# EPICS substitutions: ek9000App/Db/EL2004.substitutions
file EL2004.template
{       pattern
        {
                TERMINAL,

        }
        {
        }
}
